// SIMATIC S7-200 project (STEP 7-Micro/WIN), CPU 221 REL 01.10

SYMBOL_TABLE USER1
Start            I0.0
Stopp            I0.1
TrucA            Q0.0
TrucB            Q0.1
TrucC            Q0.2
TrucD            Q0.3
END_SYMBOL_TABLE

ORGANIZATION_BLOCK MAIN:OB1
TITLE=
BEGIN
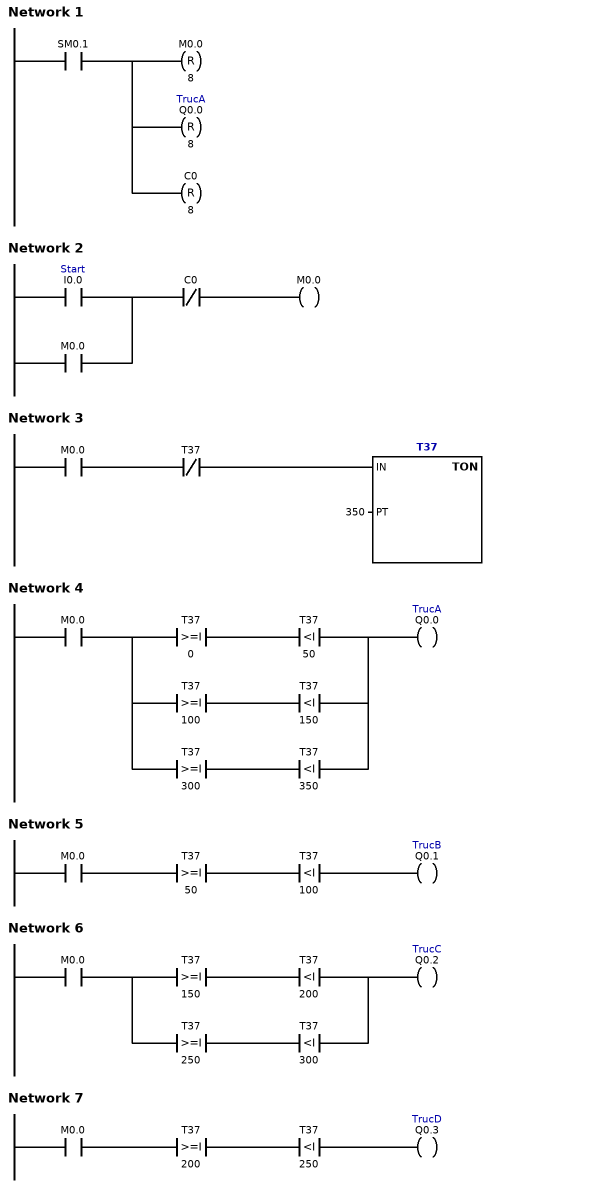
Network 1
LD     SM0.1
R      M0.0, 8
R      TrucA:Q0.0, 8
R      C0, 8
Network 2
LD     Start:I0.0
O      M0.0
AN     C0
=      M0.0
Network 3
LD     M0.0
AN     T37
TON    T37, 350
Network 4
LD     M0.0
LDW>=  T37, 0
AW<    T37, 50
LDW>=  T37, 100
AW<    T37, 150
OLD
LDW>=  T37, 300
AW<    T37, 350
OLD
ALD
=      TrucA:Q0.0
Network 5
LD     M0.0
AW>=   T37, 50
AW<    T37, 100
=      TrucB:Q0.1
Network 6
LD     M0.0
LDW>=  T37, 150
AW<    T37, 200
LDW>=  T37, 250
AW<    T37, 300
OLD
ALD
=      TrucC:Q0.2
Network 7
LD     M0.0
AW>=   T37, 200
AW<    T37, 250
=      TrucD:Q0.3
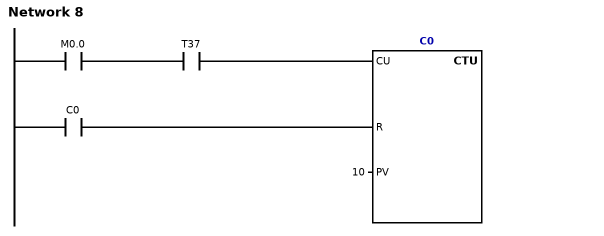
Network 8
LD     M0.0
A      T37
LD     C0
CTU    C0, 10
END_ORGANIZATION_BLOCK
